# EPICS IOC start-up script: iocsh/ethercatmcEL6688-EL1252-PTP-POS-NEG.iocsh
ethercatmcCreateAsynParam $(MOTOR_PORT) TS_NS_POS             Int32
ethercatmcCreateAsynParam $(MOTOR_PORT) TS_NS_NEG             Int32

dbLoadRecords("ethercatmcEL6688-EL1252-PTP-POS-NEG.template", "P=$(P), R=$(R), MOTOR_PORT=$(MOTOR_PORT)")
